PROGRAM P_IncDruck
VAR
END_VAR

IF DB6.rDrahthalterSchliessdruck < 5.9 THEN
	DB6.rDrahthalterSchliessdruck := DB6.rDrahthalterSchliessdruck + 0.5;
END_IF

END_PROGRAM

(* stored: Version 1.1.0.1, ProductVersion 3.1.4024.3
   POU P_IncDruck: Id {6eb67aaa-a90b-4d77-9125-dde8fd5a48c5}, SpecialFunc None *)
